FUNCTION_BLOCK Test_NotificationCountWithQueueingEnabled EXTENDS T_UnitTestBase
VAR
    Notification   : T_Notification;
    NotificationHandler : T_NotificationHandler;
    IsRaised : BOOL;
	Assertion : T_Assertion;
END_VAR

{attribute 'analysis' := '-33'} // inhibit unused variable warning
METHOD RunTest
VAR_OUTPUT
    TestCompleted : BOOL;
    TestFailed    : BOOL;
END_VAR
NotificationHandler.FB_init(bInitRetains    := FALSE,
                            bInCopyCode     := FALSE);
							
NotificationHandler.NotificationQueueingEnabled := TRUE; // Notification Queuing requires care to ensure all notifications are handled, so disabled by default!

Notification.ClearNotificationHandlers().AddNotificationHandler(NotificationHandler);

Notification.Raise();
Notification.Raise();
Notification.Raise();

TestFailed S= NOT Assertion.AssertEquals_DINT(Source       := TestName,
                                              Expected     := 3,
                                              Actual       := NotificationHandler.NotificationCount,
                                              VariableName := 'Handler.NotificationCount');

TestFailed S= NOT Assertion.AssertEquals_BOOL(Source       := TestName,
                                              Expected     := TRUE,
                                              Actual       := NotificationHandler.IsRaised(),
                                              VariableName := 'IsRaised');

TestFailed S= NOT Assertion.AssertEquals_DINT(Source       := TestName,
                                              Expected     := 2,
                                              Actual       := NotificationHandler.NotificationCount,
                                              VariableName := 'Handler.NotificationCount');

TestFailed S= NOT Assertion.AssertEquals_BOOL(Source       := TestName,
                                              Expected     := TRUE,
                                              Actual       := NotificationHandler.IsRaised(),
                                              VariableName := 'IsRaised');

TestFailed S= NOT Assertion.AssertEquals_DINT(Source       := TestName,
                                              Expected     := 1,
                                              Actual       := NotificationHandler.NotificationCount,
                                              VariableName := 'Handler.NotificationCount');

IsRaised   := NotificationHandler.IsRaised();
TestFailed S= NOT Assertion.AssertEquals_BOOL(Source       := TestName,
                                              Expected     := TRUE,
                                              Actual       := IsRaised,
                                              VariableName := 'IsRaised');

TestFailed S= NOT Assertion.AssertEquals_DINT(Source       := TestName,
                                              Expected     := 0,
                                              Actual       := NotificationHandler.NotificationCount,
                                              VariableName := 'Handler.NotificationCount');

TestFailed S= NOT Assertion.AssertEquals_BOOL(Source       := TestName,
                                              Expected     := FALSE,
                                              Actual       := NotificationHandler.IsRaised(),
                                              VariableName := 'Handler.IsRaised()');

TestCompleted := TRUE;
END_METHOD

END_FUNCTION_BLOCK

(* stored: Version 1.1.0.1, ProductVersion 3.1.4024.12
   POU Test_NotificationCountWithQueueingEnabled: Id {cc4afe9e-8e15-4d59-a92f-3d05885e6e5b}, SpecialFunc None
   Method RunTest: Id {b79fb909-26ec-4e45-bdd8-8d8681676f8c} *)
